INTERFACE IUnitTest EXTENDS __SYSTEM.IQueryInterface

METHOD Execute
END_METHOD

METHOD Initialise
VAR_INPUT
    MessageList : IAssertionMessageList;
END_VAR
END_METHOD

PROPERTY TestHasFailed : BOOL
GET
END_GET
END_PROPERTY

PROPERTY TestHasFinished : BOOL
GET
END_GET
END_PROPERTY

PROPERTY TestName : T_MaxString
GET
END_GET
END_PROPERTY

END_INTERFACE

(* stored: Version 1.1.0.1, ProductVersion 3.1.4024.4
   Itf IUnitTest: Id {5a865065-1461-4713-8b72-2d119ca0555a}
   Method Execute: Id {5b8843d7-4cda-4c26-9de3-be7fac99b2df}
   Method Initialise: Id {9fa25a66-9b79-49d4-a1db-f7754906e1ac}
   Property TestHasFailed: Id {b3492329-9de3-4a09-9fad-26085c91b577}
   Get Get: Id {86c6f866-6427-453e-89d8-c1b3ee4a7196}
   Property TestHasFinished: Id {493589bb-3ee3-4901-af36-1621c899024d}
   Get Get: Id {16cee2ab-a5b6-40b9-94d3-5031542657b0}
   Property TestName: Id {ae85e44c-4aaf-43d7-bbf9-20ebb283ad73}
   Get Get: Id {6add4a7d-7111-429c-aa26-265aa41be0d2} *)
